(* IEC 61131-3 sources: vertical-injection-machine-docs/docs/IM_SYS_PRG/Code/顶出系统/托模, 3 files *)

(* ---- EjectTypes.st ---- *)
(*
  EjectTypes.st
  功能：
  1. 定义托模基础动作和托模组合模式使用的状态枚举与参数结构。
  2. 统一托模进、保持、退以及定次/震动/停留模式的数据边界。
*)

TYPE E_EjectState :
(
    eState_Idle,         // 空闲
    eState_Init,         // 初始化
    eState_EjectIning,   // 托模进执行中
    eState_EjectIned,    // 托模进完成
    eState_EjectKeeping, // 托模保持执行中
    eState_EjectKept,    // 托模保持完成
    eState_EjectOuting,  // 托模退执行中
    eState_EjectOuted,   // 托模退完成
    eState_Error         // 故障
);
END_TYPE

TYPE ST_EjectSeg :
STRUCT
    uiPres: UINT;     // 段目标压力
    uiSpd: UINT;      // 段目标速度
    udiPos: UDINT;    // 段目标位置
    uiTime: UINT;     // 段最长执行时间
    uiPresGrad: UINT; // 压力渐进值
    uiSpdGrad: UINT;  // 速度渐进值
END_STRUCT
END_TYPE

TYPE ST_EjectPara :
STRUCT
    uiEjectInSegCnt: UINT;                     // 托模进段数量
    uiEjectInMode: UINT;                       // 托模进控制模式
    uiEjectInLimitTime: UINT;                  // 托模进最大允许时间
    aEjectInSeg: ARRAY[1..3] OF ST_EjectSeg;   // 托模进段参数
    uiEjectInPresStartGrad: UINT;              // 托模进压力起始渐进
    uiEjectInPresStopGrad: UINT;               // 托模进压力停止渐进
    uiEjectInSpdStartGrad: UINT;               // 托模进速度起始渐进
    uiEjectInSpdStopGrad: UINT;                // 托模进速度停止渐进
    stEjectKeepSeg: ST_EjectSeg;               // 托模保持段参数
    uiEjectOutSegCnt: UINT;                    // 托模退段数量
    uiEjectOutMode: UINT;                      // 托模退控制模式
    uiEjectOutLimitTime: UINT;                 // 托模退最大允许时间
    aEjectOutSeg: ARRAY[1..3] OF ST_EjectSeg;  // 托模退段参数
    uiEjectOutPresStartGrad: UINT;             // 托模退压力起始渐进
    uiEjectOutPresStopGrad: UINT;              // 托模退压力停止渐进
    uiEjectOutSpdStartGrad: UINT;              // 托模退速度起始渐进
    uiEjectOutSpdStopGrad: UINT;               // 托模退速度停止渐进
    stEjectInDbgSeg: ST_EjectSeg;              // 托模进调试段参数
    stEjectOutDbgSeg: ST_EjectSeg;             // 托模退调试段参数
END_STRUCT
END_TYPE

TYPE E_EjectModeState :
(
    eState_Idle,       // 空闲
    eState_Init,       // 初始化
    eState_EjectCount, // 定次托模模式
    eState_EjectVibra, // 震动托模模式
    eState_EjectHold,  // 停留托模模式
    eState_Error       // 故障
);
END_TYPE

(* ---- FB_Eject.st ---- *)
(*
  FB_Eject 功能块
  功能：
  1. 负责托模进、托模保持、托模退及其调试动作的执行状态机。
  2. 按托模参数输出压力、速度、位置命令，并返回托模进退完成状态。

  说明：
  1. 正常模式使用 1=托模进、2=托模退；调试模式使用 6/7。
  2. 组合托模模式由 `FB_EjectMode` 复用本块完成具体动作。
*)
FUNCTION_BLOCK FB_Eject
VAR_IN_OUT
    stEjectAxis: ST_AxisRefHyd;       // 托模共享轴结构
END_VAR
VAR_INPUT
    bStart: BOOL;                     // TRUE=启动托模动作
    bStop: BOOL;                      // TRUE=正常停止
    bEStop: BOOL;                     // TRUE=急停
    bReset: BOOL;                     // TRUE=复位状态机与输出
    bManualMode: BOOL;                // TRUE=手动点动托模
    uiEjectMode: UINT;                // 1=托模进 2=托模退 6=托模进调试 7=托模退调试
    stEjectPara: ST_EjectPara;        // 托模工艺参数
    bEjectInStop: BOOL;               // 托模进停止信号
    bEjectOutStop: BOOL;              // 托模退停止信号
    udiEjectElecRulerVal: UDINT;      // 位置反馈
    rEjectActualPosition: LREAL;      // 托模轴实际位置反馈
    rEjectActualVelocity: LREAL;      // 托模轴实际速度反馈
    rEjectActualPressure: LREAL;      // 托模轴实际压力反馈
END_VAR
VAR_OUTPUT
    bBusy: BOOL;                      // TRUE=当前动作尚未结束
    bDone: BOOL;                      // TRUE=当前动作完成
    bAlarm: BOOL;                     // TRUE=当前动作报警
    dwAlarmID: DWORD;                 // 模块报警码
    uiActHint: UINT;                  // 当前动作提示码
    uiActTime: UINT;                  // 当前动作持续时间，单位 s
    bEjectIned: BOOL;                 // TRUE=托模进完成
    bEjectOuted: BOOL;                // TRUE=托模退完成
    uiPresCmd: UINT;                  // 压力命令输出
    uiSpdCmd: UINT;                   // 速度命令输出
    udiPosCmd: UDINT;                 // 位置命令输出
END_VAR
VAR
    eState: E_EjectState := eState_Idle; // 当前托模状态机状态
    fbAxisInst: FB_HydAxis;              // 托模轴层实例
    stAxisStatusLocal: ST_HydAxisStatus; // 托模轴层状态缓存
    stAxisConfigLocal: ST_HydAxisConfig := (
        nAxisID := 6,
        rMaxCylinderStroke := 10000.0,
        rMaxVelocity := 1000.0,
        rMaxPressure := 1000.0,
        rPosTolerance := 0.5,
        rVelTolerance := 0.5,
        rPresTolerance := 0.5
    );
    uiStageIndex: UINT := 0;             // 当前执行到的托模进/托模退段号
    tPulse: TON;                         // 100ms 节拍定时器，用于累计动作时间
    udiElapsedMs: UDINT := 0;            // 当前托模动作或保持段已运行时间，单位 ms
    bManualActive: BOOL := FALSE;        // TRUE=当前按调试/手动逻辑执行
    bInRequest: BOOL := FALSE;           // TRUE=当前请求方向为托模进
    bOutRequest: BOOL := FALSE;          // TRUE=当前请求方向为托模退
    stSegCmd: ST_EjectSeg;               // 当前生效的托模段命令缓存
END_VAR

(* 每拍先把模式号映射成统一的托进/托退/手动语义。 *)
bManualActive := bManualMode OR (uiEjectMode = 6) OR (uiEjectMode = 7);
bInRequest := (uiEjectMode = 1) OR (uiEjectMode = 6);
bOutRequest := (uiEjectMode = 2) OR (uiEjectMode = 7);

(* 复位优先级最高：清空完成态、段号、计时和输出命令。 *)
IF bReset THEN
    eState := eState_Idle;
    bBusy := FALSE;
    bDone := FALSE;
    bAlarm := FALSE;
    dwAlarmID := 0;
    uiActHint := 0;
    uiActTime := 0;
    bEjectIned := FALSE;
    bEjectOuted := FALSE;
    uiPresCmd := 0;
    uiSpdCmd := 0;
    udiPosCmd := 0;
    uiStageIndex := 0;
    udiElapsedMs := 0;
    tPulse(IN := FALSE, PT := T#100MS);
(* 急停直接转故障态，立即撤销托模命令。 *)
ELSIF bEStop THEN
    eState := eState_Error;
    bAlarm := TRUE;
    dwAlarmID := dwAlarmID OR DWORD#16#0010;
    uiActHint := 1;
    uiPresCmd := 0;
    uiSpdCmd := 0;
    udiPosCmd := 0;
    tPulse(IN := FALSE, PT := T#100MS);
(* 正常停止按空闲态收口，等待重新启动。 *)
ELSIF bStop THEN
    eState := eState_Idle;
    bBusy := FALSE;
    uiPresCmd := 0;
    uiSpdCmd := 0;
    udiPosCmd := 0;
    uiActHint := 0;
    udiElapsedMs := 0;
    tPulse(IN := FALSE, PT := T#100MS);
ELSE
    CASE eState OF
        (* 空闲态：等待启动，并根据请求方向进入托模进或托模退。 *)
        eState_Idle:
            bBusy := FALSE;
            bDone := FALSE;
            uiActHint := 0;
            uiActTime := 0;
            bEjectIned := FALSE;
            bEjectOuted := FALSE;
            uiPresCmd := 0;
            uiSpdCmd := 0;
            udiPosCmd := 0;
            uiStageIndex := 0;
            udiElapsedMs := 0;
            tPulse(IN := FALSE, PT := T#100MS);
            IF bStart THEN
                bAlarm := FALSE;
                dwAlarmID := 0;
                uiStageIndex := 1;
                IF bInRequest THEN
                    eState := eState_EjectIning;
                ELSIF bOutRequest THEN
                    eState := eState_EjectOuting;
                ELSE
                    bAlarm := TRUE;
                    dwAlarmID := DWORD#16#0001;
                    eState := eState_Error;
                END_IF;
            END_IF;

        (* 托模进执行态：自动模式按段推进，手动模式持续输出调试段。 *)
        eState_EjectIning:
            bBusy := TRUE;
            tPulse(IN := TRUE, PT := T#100MS);
            IF tPulse.Q THEN
                udiElapsedMs := udiElapsedMs + 100;
                tPulse(IN := FALSE, PT := T#100MS);
            END_IF;
            uiActTime := TO_UINT(udiElapsedMs / 1000);

            (* 调试托模进优先使用调试段；未配置时回退到正式第一段。 *)
            IF bManualActive THEN
                stSegCmd := stEjectPara.stEjectInDbgSeg;
                IF (stSegCmd.uiPres = 0) AND (stSegCmd.uiSpd = 0) AND (stSegCmd.udiPos = 0) THEN
                    stSegCmd := stEjectPara.aEjectInSeg[1];
                END_IF;
                uiActHint := 28;
                uiPresCmd := stSegCmd.uiPres;
                uiSpdCmd := stSegCmd.uiSpd;
                udiPosCmd := stSegCmd.udiPos;
                IF NOT bStart THEN
                    eState := eState_Idle;
                END_IF;
            (* 自动托模进按段执行。所有前进段结束后，视配置决定是否进入托模保持。 *)
            ELSE
                IF uiStageIndex > stEjectPara.uiEjectInSegCnt THEN
                    IF stEjectPara.stEjectKeepSeg.uiTime > 0 THEN
                        eState := eState_EjectKeeping;
                    ELSE
                        eState := eState_EjectIned;
                    END_IF;
                    udiElapsedMs := 0;
                    tPulse(IN := FALSE, PT := T#100MS);
                ELSE
                    stSegCmd := stEjectPara.aEjectInSeg[uiStageIndex];
                    uiActHint := 89 + uiStageIndex; // 90-92
                    uiPresCmd := stSegCmd.uiPres;
                    uiSpdCmd := stSegCmd.uiSpd;
                    udiPosCmd := stSegCmd.udiPos;

                    (* `uiEjectInMode` 约定：
                       0=按段时间推进；
                       1=按托模进停止信号推进；
                       2=按电子尺位置推进。 *)
                    IF (stEjectPara.uiEjectInMode = 2) AND (udiEjectElecRulerVal >= stSegCmd.udiPos) THEN
                        uiStageIndex := uiStageIndex + 1;
                        udiElapsedMs := 0;
                        tPulse(IN := FALSE, PT := T#100MS);
                    ELSIF ((stEjectPara.uiEjectInMode = 0) AND (stSegCmd.uiTime > 0) AND (udiElapsedMs >= TO_UDINT(stSegCmd.uiTime))) OR ((stEjectPara.uiEjectInMode = 1) AND bEjectInStop) THEN
                        uiStageIndex := uiStageIndex + 1;
                        udiElapsedMs := 0;
                        tPulse(IN := FALSE, PT := T#100MS);
                    END_IF;

                    (* 托模进总时长超限后直接报警。 *)
                    IF (stEjectPara.uiEjectInLimitTime > 0) AND (udiElapsedMs >= TO_UDINT(stEjectPara.uiEjectInLimitTime)) THEN
                        dwAlarmID := dwAlarmID OR DWORD#16#0001;
                        eState := eState_Error;
                    END_IF;
                END_IF;
            END_IF;

        (* 托模进完成态：对外发布“托模进完成”。 *)
        eState_EjectIned:
            bBusy := FALSE;
            bDone := TRUE;
            bEjectIned := TRUE;
            uiActHint := 30;
            uiPresCmd := 0;
            uiSpdCmd := 0;
            udiPosCmd := 0;

        (* 托模保持态：用独立保持段在当前位置维持压力/速度设定。 *)
        eState_EjectKeeping:
            bBusy := TRUE;
            uiActHint := 29;
            uiPresCmd := stEjectPara.stEjectKeepSeg.uiPres;
            uiSpdCmd := stEjectPara.stEjectKeepSeg.uiSpd;
            udiPosCmd := stEjectPara.stEjectKeepSeg.udiPos;
            tPulse(IN := TRUE, PT := T#100MS);
            IF tPulse.Q THEN
                udiElapsedMs := udiElapsedMs + 100;
                tPulse(IN := FALSE, PT := T#100MS);
            END_IF;
            uiActTime := TO_UINT(udiElapsedMs / 1000);
            (* 保持时间到后转入“已保持”完成态；时间为 0 则本拍立即完成。 *)
            IF (stEjectPara.stEjectKeepSeg.uiTime = 0) OR (udiElapsedMs >= TO_UDINT(stEjectPara.stEjectKeepSeg.uiTime)) THEN
                eState := eState_EjectKept;
                tPulse(IN := FALSE, PT := T#100MS);
            END_IF;

        (* 托模保持完成态：对外仍以“托模进完成”语义对接上层。 *)
        eState_EjectKept:
            bBusy := FALSE;
            bDone := TRUE;
            bEjectIned := TRUE;
            uiActHint := 29;
            uiPresCmd := 0;
            uiSpdCmd := 0;
            udiPosCmd := 0;

        (* 托模退执行态：自动模式按段推进，手动模式持续输出调试段。 *)
        eState_EjectOuting:
            bBusy := TRUE;
            tPulse(IN := TRUE, PT := T#100MS);
            IF tPulse.Q THEN
                udiElapsedMs := udiElapsedMs + 100;
                tPulse(IN := FALSE, PT := T#100MS);
            END_IF;
            uiActTime := TO_UINT(udiElapsedMs / 1000);

            (* 调试托模退优先使用调试段；未配置时回退到正式第一段。 *)
            IF bManualActive THEN
                stSegCmd := stEjectPara.stEjectOutDbgSeg;
                IF (stSegCmd.uiPres = 0) AND (stSegCmd.uiSpd = 0) AND (stSegCmd.udiPos = 0) THEN
                    stSegCmd := stEjectPara.aEjectOutSeg[1];
                END_IF;
                uiActHint := 31;
                uiPresCmd := stSegCmd.uiPres;
                uiSpdCmd := stSegCmd.uiSpd;
                udiPosCmd := stSegCmd.udiPos;
                IF NOT bStart THEN
                    eState := eState_Idle;
                END_IF;
            (* 自动托模退按段执行，完成条件支持位置、停止信号或时间。 *)
            ELSE
                IF uiStageIndex > stEjectPara.uiEjectOutSegCnt THEN
                    eState := eState_EjectOuted;
                ELSE
                    stSegCmd := stEjectPara.aEjectOutSeg[uiStageIndex];
                    uiActHint := 91 + uiStageIndex; // 92-94
                    uiPresCmd := stSegCmd.uiPres;
                    uiSpdCmd := stSegCmd.uiSpd;
                    udiPosCmd := stSegCmd.udiPos;

                    (* `uiEjectOutMode` 约定：
                       0=按段时间推进；
                       1=按托模退停止信号推进；
                       2=按电子尺位置推进。 *)
                    IF (stEjectPara.uiEjectOutMode = 2) AND (udiEjectElecRulerVal >= stSegCmd.udiPos) THEN
                        uiStageIndex := uiStageIndex + 1;
                        udiElapsedMs := 0;
                        tPulse(IN := FALSE, PT := T#100MS);
                    ELSIF ((stEjectPara.uiEjectOutMode = 0) AND (stSegCmd.uiTime > 0) AND (udiElapsedMs >= TO_UDINT(stSegCmd.uiTime))) OR ((stEjectPara.uiEjectOutMode = 1) AND bEjectOutStop) THEN
                        uiStageIndex := uiStageIndex + 1;
                        udiElapsedMs := 0;
                        tPulse(IN := FALSE, PT := T#100MS);
                    END_IF;

                    (* 托模退总时长超限时直接报警。 *)
                    IF (stEjectPara.uiEjectOutLimitTime > 0) AND (udiElapsedMs >= TO_UDINT(stEjectPara.uiEjectOutLimitTime)) THEN
                        dwAlarmID := dwAlarmID OR DWORD#16#0002;
                        eState := eState_Error;
                    END_IF;
                END_IF;
            END_IF;

        (* 托模退完成态：置位托模退完成标志。 *)
        eState_EjectOuted:
            bBusy := FALSE;
            bDone := TRUE;
            bEjectOuted := TRUE;
            uiActHint := 32;
            uiPresCmd := 0;
            uiSpdCmd := 0;
            udiPosCmd := 0;

        (* 故障态：统一撤销托模输出，仅保留报警。 *)
        eState_Error:
            bBusy := FALSE;
            bAlarm := TRUE;
            uiActHint := 1;
            uiPresCmd := 0;
            uiSpdCmd := 0;
            udiPosCmd := 0;
            tPulse(IN := FALSE, PT := T#100MS);

    ELSE
        eState := eState_Error;
    END_CASE;
END_IF;

(* 先把现场反馈、固定轴配置和模块报警写回共享轴结构，再通过统一轴层接口下发托模命令。 *)
stEjectAxis.rActualPosition := rEjectActualPosition;
stEjectAxis.rActualVelocity := rEjectActualVelocity;
stEjectAxis.rActualPressure := rEjectActualPressure;
stEjectAxis.stConfig := stAxisConfigLocal;
stEjectAxis.nFaultCode := TO_INT(dwAlarmID);

fbAxisInst(
    stAxisRef := stEjectAxis,        // 把托模共享轴结构交给轴层实例统一整理最终命令与状态。
    bStart := bBusy,                 // 托模模块当前忙碌时，通知轴层继续执行本拍目标命令。
    bStop := bStop,                  // 把托模模块收到的正常停止命令直接送给轴层。
    bEStop := bEStop,                // 把托模模块收到的急停命令直接送给轴层。
    bReset := bReset,                // 把托模模块收到的复位命令直接送给轴层。
    bDir := bInRequest,              // 当前把“TRUE=托模进方向”定义为托模轴正向方向。
    uiMode := UINT#1,                // 当前液压执行链统一按位置模式接口收口。
    uiCmdPres := uiPresCmd,          // 把托模模块当前压力命令送给轴层做最终压力限幅。
    uiSpd := uiSpdCmd,               // 把托模模块当前速度命令送给轴层做最终速度限幅。
    udiPos := udiPosCmd,             // 把托模模块当前位置目标送给轴层做最终行程限幅。
    uiForce := UINT#0,               // 当前托模模块未定义独立力命令，因此该接口位先固定传 0。
    uiAcc := UINT#0,                 // 当前托模模块未定义独立加速度命令，因此该接口位先固定传 0。
    uiDec := UINT#0,                 // 当前托模模块未定义独立减速度命令，因此该接口位先固定传 0。
    uiJerk := UINT#0                 // 当前托模模块未定义独立加加速度命令，因此该接口位先固定传 0。
);

stAxisStatusLocal := stEjectAxis.stStatus; // 把共享轴结构中的轴层状态镜像到模块本地缓存，沿用现有汇总代码。

bBusy := bBusy OR stAxisStatusLocal.bCommandActive;
bAlarm := bAlarm OR stAxisStatusLocal.bAlarm;
dwAlarmID := dwAlarmID OR stAxisStatusLocal.dwAlarmID;
IF stAxisStatusLocal.uiActTime > uiActTime THEN
    uiActTime := stAxisStatusLocal.uiActTime;
END_IF;
END_FUNCTION_BLOCK

(* ---- FB_EjectMode.st ---- *)
(*
  FB_EjectMode 功能块
  功能：
  1. 在基础 `FB_Eject` 之上组合出定次、震动、停留三种托模模式。
  2. 通过内部顺序控制，把“托模进/托模退/托模保持”拼成更高层动作。
  3. 对外仍保持与普通托模模块相似的 Busy/Done/Alarm 接口，便于主控统一调用。

  说明：
  1. 本块本身不直接生成液压命令，而是复用 `FB_Eject` 完成具体动作。
  2. `uiSeqPhase` 用来表示当前执行到“复位子块、托进、再次复位、托退”的哪一步。
  3. 只有在手动组合模式被上层明确选择时，才应该让本块接管托模轴输出。
*)
FUNCTION_BLOCK FB_EjectMode
VAR_IN_OUT
    stEjectAxis: ST_AxisRefHyd;   // 托模共享轴结构，内部复用的 `FB_Eject` 直接操作该轴
END_VAR
VAR_INPUT
    bStart: BOOL;                 // TRUE=启动组合托模模式
    bStop: BOOL;                  // TRUE=正常停止当前组合流程
    bEStop: BOOL;                 // TRUE=急停，立即撤销对子块的命令
    bReset: BOOL;                 // TRUE=复位本块及内部 `FB_Eject`
    uiEjectMode: UINT;            // 1=定次 2=震动 3=停留
    uiEjectTimes: UINT;           // 定次/震动次数；震动模式下 0 表示持续循环
    stEjectPara: ST_EjectPara;    // 传给内部 `FB_Eject` 的托模工艺参数
    bEjectInStop: BOOL;           // 托模进停止信号，直接透传给内部 `FB_Eject`
    bEjectOutStop: BOOL;          // 托模退停止信号，直接透传给内部 `FB_Eject`
    udiEjectElecRulerVal: UDINT;  // 托模电子尺反馈，直接透传给内部 `FB_Eject`
END_VAR
VAR_OUTPUT
    bBusy: BOOL;                  // TRUE=组合托模模式尚未完成
    bDone: BOOL;                  // TRUE=组合托模模式完成
    bAlarm: BOOL;                 // TRUE=本块或内部 `FB_Eject` 报警
    dwAlarmID: DWORD;             // 组合块报警码，优先透传子块报警
    uiActHint: UINT;              // 当前动作提示码，默认复用子块提示
    uiActTime: UINT;              // 当前动作持续时间，默认复用子块计时
    bEjectIned: BOOL;             // TRUE=内部托模进完成
    bEjectOuted: BOOL;            // TRUE=内部托模退完成
    uiPresCmd: UINT;              // 当前对子块输出的压力命令镜像
    uiSpdCmd: UINT;               // 当前对子块输出的速度命令镜像
    udiPosCmd: UDINT;             // 当前对子块输出的位置命令镜像
END_VAR
VAR
    eState: E_EjectModeState := eState_Idle; // 当前组合托模状态机状态
    fbEject: FB_Eject;                       // 内部基础托模块实例，实际液压命令由它生成

    (* 发给内部 `FB_Eject` 的命令。 *)
    bCmdStart: BOOL := FALSE;               // TRUE=本拍触发内部 `FB_Eject` 启动
    bCmdReset: BOOL := FALSE;               // TRUE=本拍复位内部 `FB_Eject`
    uiCmdMode: UINT := 0;                   // 发给内部 `FB_Eject` 的模式号，1=托进 2=托退

    (* 顺序控制变量。 *)
    uiExecCount: UINT := 0;                 // 已完成的往返或震动次数
    uiSeqPhase: UINT := 0;                  // 当前子流程相位：0复位前置 1托进 2退前复位 3托退

    (* 内部 `FB_Eject` 状态缓存。 *)
    bSubBusy: BOOL := FALSE;                // 内部 `FB_Eject` Busy 状态缓存
    bSubDone: BOOL := FALSE;                // 内部 `FB_Eject` Done 状态缓存
    bSubAlarm: BOOL := FALSE;               // 内部 `FB_Eject` Alarm 状态缓存
    dwSubAlarmID: DWORD := 0;               // 内部 `FB_Eject` 报警码缓存
    uiSubActHint: UINT := 0;                // 内部 `FB_Eject` 当前动作提示缓存
    uiSubActTime: UINT := 0;                // 内部 `FB_Eject` 当前动作时间缓存
    bSubEjectIned: BOOL := FALSE;           // 内部 `FB_Eject` 托模进完成缓存
    bSubEjectOuted: BOOL := FALSE;          // 内部 `FB_Eject` 托模退完成缓存
    uiSubPresCmd: UINT := 0;                // 内部 `FB_Eject` 压力命令缓存
    uiSubSpdCmd: UINT := 0;                 // 内部 `FB_Eject` 速度命令缓存
    udiSubPosCmd: UDINT := 0;               // 内部 `FB_Eject` 位置命令缓存
END_VAR

(* 每个扫描周期先清空对子块的控制命令。 *)
bCmdStart := FALSE;
bCmdReset := FALSE;
uiCmdMode := 0;

(* 复位优先级最高：本块回空闲，同时给内部子块打一拍复位。 *)
IF bReset THEN
    eState := eState_Idle;
    bBusy := FALSE;
    bDone := FALSE;
    bAlarm := FALSE;
    dwAlarmID := DWORD#0;
    uiActHint := 0;
    uiActTime := 0;
    uiExecCount := 0;
    uiSeqPhase := 0;
    bCmdReset := TRUE;

(* 急停直接转故障态，并强制复位子块，确保托模轴命令被撤销。 *)
ELSIF bEStop THEN
    eState := eState_Error;
    bBusy := FALSE;
    bDone := FALSE;
    bAlarm := TRUE;
    dwAlarmID := DWORD#16#0010;
    uiActHint := 1;
    uiActTime := 0;
    uiExecCount := 0;
    uiSeqPhase := 0;
    bCmdReset := TRUE;

(* 正常停止直接回空闲，同样复位子块，避免保留上一个动作的完成态。 *)
ELSIF bStop THEN
    eState := eState_Idle;
    bBusy := FALSE;
    bDone := FALSE;
    bAlarm := FALSE;
    dwAlarmID := DWORD#0;
    uiActHint := 0;
    uiActTime := 0;
    uiExecCount := 0;
    uiSeqPhase := 0;
    bCmdReset := TRUE;

ELSE
    CASE eState OF
        (* 空闲态：等待启动，并按组合模式切入定次、震动或停留逻辑。 *)
        eState_Idle:
            bBusy := FALSE;
            uiActHint := 0;
            uiActTime := 0;

            IF bStart THEN
                bDone := FALSE;
                bAlarm := FALSE;
                dwAlarmID := DWORD#0;
                uiExecCount := 0;
                uiSeqPhase := 0;

                CASE uiEjectMode OF
                    1: eState := eState_EjectCount;
                    2: eState := eState_EjectVibra;
                    3: eState := eState_EjectHold;
                ELSE
                    bAlarm := TRUE;
                    dwAlarmID := DWORD#16#0001;
                    eState := eState_Error;
                END_CASE;
            END_IF;

        (* 定次托模态：按“托进 -> 托退”为一个完整循环，达到次数后结束。 *)
        eState_EjectCount:
            bBusy := TRUE;

            IF bSubAlarm THEN
                dwAlarmID := dwSubAlarmID;
                eState := eState_Error;
            ELSE
                (* `uiSeqPhase` 把一个往返拆成“复位子块、托进、再次复位、托退”四步。 *)
                CASE uiSeqPhase OF
                    0:
                        (* 子块切换动作前先复位，避免沿用上一个动作的完成态。 *)
                        bCmdReset := TRUE;
                        uiSeqPhase := 1;

                    1:
                        (* 托模进。 *)
                        uiCmdMode := 1;
                        bCmdStart := TRUE;
                        IF bSubDone THEN
                            uiSeqPhase := 2;
                        END_IF;

                    2:
                        (* 进入托模退前再复位一次子块。 *)
                        bCmdReset := TRUE;
                        uiSeqPhase := 3;

                    3:
                        (* 托模退。 *)
                        uiCmdMode := 2;
                        bCmdStart := TRUE;
                        IF bSubDone THEN
                            uiExecCount := uiExecCount + 1;
                            (* 定次模式下 `uiEjectTimes = 0` 仍按 1 次收口，避免无终点循环。 *)
                            IF uiExecCount >= SEL(uiEjectTimes = 0, uiEjectTimes, 1) THEN
                                bBusy := FALSE;
                                bDone := TRUE;
                                eState := eState_Idle;
                            ELSE
                                uiSeqPhase := 0;
                            END_IF;
                        END_IF;

                ELSE
                    uiSeqPhase := 0;
                END_CASE;
            END_IF;

        (* 震动态：同样执行“托进 -> 托退”循环，但 `uiEjectTimes = 0` 表示持续循环。 *)
        eState_EjectVibra:
            bBusy := TRUE;

            IF bSubAlarm THEN
                dwAlarmID := dwSubAlarmID;
                eState := eState_Error;
            ELSE
                (* 相位定义与定次模式一致，只是结束条件不同。 *)
                CASE uiSeqPhase OF
                    0:
                        bCmdReset := TRUE;
                        uiSeqPhase := 1;

                    1:
                        uiCmdMode := 1;
                        bCmdStart := TRUE;
                        IF bSubDone THEN
                            uiSeqPhase := 2;
                        END_IF;

                    2:
                        bCmdReset := TRUE;
                        uiSeqPhase := 3;

                    3:
                        uiCmdMode := 2;
                        bCmdStart := TRUE;
                        IF bSubDone THEN
                            uiExecCount := uiExecCount + 1;
                            IF (uiEjectTimes > 0) AND (uiExecCount >= uiEjectTimes) THEN
                                bBusy := FALSE;
                                bDone := TRUE;
                                eState := eState_Idle;
                            ELSE
                                uiSeqPhase := 0;
                            END_IF;
                        END_IF;

                ELSE
                    uiSeqPhase := 0;
                END_CASE;
            END_IF;

        (* 停留态：只执行一次托模进，完成后停在前进端。 *)
        eState_EjectHold:
            bBusy := TRUE;

            IF bSubAlarm THEN
                dwAlarmID := dwSubAlarmID;
                eState := eState_Error;
            ELSE
                (* 停留模式只需要“复位子块 -> 托进”两个步骤。 *)
                CASE uiSeqPhase OF
                    0:
                        bCmdReset := TRUE;
                        uiSeqPhase := 1;

                    1:
                        uiCmdMode := 1;
                        bCmdStart := TRUE;
                        IF bSubDone THEN
                            bBusy := FALSE;
                            bDone := TRUE;
                            eState := eState_Idle;
                        END_IF;

                ELSE
                    uiSeqPhase := 0;
                END_CASE;
            END_IF;

        (* 故障态：统一复位子块，并保留报警信息给主控/HMI。 *)
        eState_Error:
            bBusy := FALSE;
            bDone := FALSE;
            bAlarm := TRUE;
            uiActHint := 1;
            IF dwAlarmID = DWORD#0 THEN
                dwAlarmID := SEL(dwSubAlarmID = DWORD#0, dwSubAlarmID, DWORD#16#0001);
            END_IF;
            bCmdReset := TRUE;

    ELSE
        dwAlarmID := DWORD#16#7FFF;
        eState := eState_Error;
    END_CASE;
END_IF;

(* 最后再调用内部子块，这样本扫描周期内刚决策出来的命令能立即送到子块。 *)
fbEject(
    stEjectAxis := stEjectAxis,
    bStart := bCmdStart,
    bStop := FALSE,
    bEStop := FALSE,
    bReset := bCmdReset,
    bManualMode := FALSE,
    uiEjectMode := uiCmdMode,
    stEjectPara := stEjectPara,
    bEjectInStop := bEjectInStop,
    bEjectOutStop := bEjectOutStop,
    udiEjectElecRulerVal := udiEjectElecRulerVal,
    bBusy => bSubBusy,
    bDone => bSubDone,
    bAlarm => bSubAlarm,
    dwAlarmID => dwSubAlarmID,
    uiActHint => uiSubActHint,
    uiActTime => uiSubActTime,
    bEjectIned => bSubEjectIned,
    bEjectOuted => bSubEjectOuted,
    uiPresCmd => uiSubPresCmd,
    uiSpdCmd => uiSubSpdCmd,
    udiPosCmd => udiSubPosCmd
);

(* 对外透传内部托模块的实际动作输出，便于主控统一读取。 *)
bEjectIned := bSubEjectIned;
bEjectOuted := bSubEjectOuted;
uiPresCmd := uiSubPresCmd;
uiSpdCmd := uiSubSpdCmd;
udiPosCmd := udiSubPosCmd;

(* 未报警时优先显示子块动作提示，让外部看到当前托进/托退所在步骤。 *)
IF (NOT bAlarm) AND (uiSubActHint <> 0) THEN
    uiActHint := uiSubActHint;
END_IF;
uiActTime := uiSubActTime;
END_FUNCTION_BLOCK
